(* IEC 61131-3 sources: festo-codesys-mcp/knowledge/library/motion, 4 files *)

(* ---- FB_AxisScaler.st ---- *)
(* =============================================================
   FB_AxisScaler — Axis Unit Conversion (mm/pulses, mm-s/Hz)

   Category:     Motion
   Platform:     CODESYS V3.5 (IEC 61131-3)
   Version:      1.0
   Dependencies: None (standard IEC only)

   Converts between user units (mm, degrees) and machine units
   (encoder pulses, frequency Hz). Handles gear ratio and
   lead screw pitch calculations.

   Usage:
     fbScaler : FB_AxisScaler;
     fbScaler(rPitch := 5.0, nPulsesPerRev := 10000, rGearRatio := 1.0);
     nPulses := fbScaler.fnPosToPulses(rPositionMm := 100.0);
     rMm     := fbScaler.fnPulsesToPos(nPulses := 200000);
   ============================================================= *)
FUNCTION_BLOCK FB_AxisScaler
VAR_INPUT
    rPitch          : REAL := 5.0;         (* Lead screw pitch [mm/rev] or [deg/rev] *)
    nPulsesPerRev   : DINT := 10000;       (* Encoder pulses per revolution *)
    rGearRatio      : REAL := 1.0;         (* Gear ratio (motor/load) *)
END_VAR
VAR_OUTPUT
    rMmPerPulse     : REAL;                (* Conversion factor: mm per pulse *)
    rPulsesPerMm    : REAL;                (* Conversion factor: pulses per mm *)
END_VAR

(* Calculate conversion factors *)
IF nPulsesPerRev > 0 AND ABS(rGearRatio) > 0.0001 THEN
    rMmPerPulse := rPitch / (DINT_TO_REAL(nPulsesPerRev) * rGearRatio);
    IF ABS(rMmPerPulse) > 0.0 THEN
        rPulsesPerMm := 1.0 / rMmPerPulse;
    ELSE
        rPulsesPerMm := 0.0;
    END_IF
ELSE
    rMmPerPulse := 0.0;
    rPulsesPerMm := 0.0;
END_IF

END_FUNCTION_BLOCK

(* ---- FB_BrakeMotor.st ---- *)
(* =============================================================
   FB_BrakeMotor — Motor with Electromagnetic Brake

   Category:     Motion
   Platform:     CODESYS V3.5 (IEC 61131-3)
   Version:      1.0
   Dependencies: None (standard IEC only)

   Controls a motor with electromagnetic holding brake.
   Sequence: Release brake → wait → start motor (and reverse on stop).
   Prevents mechanical shock from simultaneous brake/motor switching.

   Usage:
     fbHoist : FB_BrakeMotor;
     fbHoist(bStart := bCmdHoist, bOverload := bDI_HoistOL);
     bMotorOut := fbHoist.bContactor;
     bBrakeOut := fbHoist.bBrakeRelease;
   ============================================================= *)
FUNCTION_BLOCK FB_BrakeMotor
VAR_INPUT
    bStart          : BOOL;                (* Start command *)
    bOverload       : BOOL := TRUE;        (* Thermal overload (NC) *)
    tBrakeDelay     : TIME := T#300MS;     (* Brake release delay before motor start *)
    tBrakeApply     : TIME := T#200MS;     (* Motor stop delay before brake apply *)
    bEnable         : BOOL := TRUE;        (* Enable control *)
    bReset          : BOOL;                (* Reset error *)
END_VAR
VAR_OUTPUT
    bContactor      : BOOL;                (* Motor contactor output *)
    bBrakeRelease   : BOOL;                (* Brake release output (TRUE=released) *)
    bRunning        : BOOL;                (* Motor is running *)
    bErr          : BOOL;                (* Error active *)
    nErrId          : DINT;                (* 0=OK, 1=Overload *)
END_VAR
VAR
    nState          : INT := 0;
    tonBrakeRel     : TON;
    tonBrakeApp     : TON;
END_VAR

(* Reset *)
IF bReset AND bErr THEN
    nState := 0;
    bErr := FALSE;
    nErrId := 0;
END_IF

(* Overload — immediate stop *)
IF NOT bOverload THEN
    bContactor := FALSE;
    bBrakeRelease := FALSE;
    bRunning := FALSE;
    bErr := TRUE;
    nErrId := 1;
    nState := 10;
    RETURN;
END_IF

IF NOT bEnable THEN
    bContactor := FALSE;
    bBrakeRelease := FALSE;
    bRunning := FALSE;
    nState := 0;
    RETURN;
END_IF

CASE nState OF
0: (* Stopped — brake applied *)
    bContactor := FALSE;
    bBrakeRelease := FALSE;
    bRunning := FALSE;
    tonBrakeRel(IN := FALSE, PT := tBrakeDelay);
    tonBrakeApp(IN := FALSE, PT := tBrakeApply);

    IF bStart THEN
        nState := 1;
    END_IF

1: (* Releasing brake *)
    bBrakeRelease := TRUE;
    bContactor := FALSE;
    tonBrakeRel(IN := TRUE, PT := tBrakeDelay);

    IF tonBrakeRel.Q THEN
        nState := 2;
        tonBrakeRel(IN := FALSE, PT := tBrakeDelay);
    END_IF

    IF NOT bStart THEN
        nState := 0;
        bBrakeRelease := FALSE;
    END_IF

2: (* Running *)
    bContactor := TRUE;
    bBrakeRelease := TRUE;
    bRunning := TRUE;

    IF NOT bStart THEN
        nState := 3;
    END_IF

3: (* Stopping — motor off, brake delayed *)
    bContactor := FALSE;
    bBrakeRelease := TRUE;
    bRunning := FALSE;
    tonBrakeApp(IN := TRUE, PT := tBrakeApply);

    IF tonBrakeApp.Q THEN
        bBrakeRelease := FALSE;
        tonBrakeApp(IN := FALSE, PT := tBrakeApply);
        nState := 0;
    END_IF

10: (* Error *)
    bContactor := FALSE;
    bBrakeRelease := FALSE;
    bRunning := FALSE;

END_CASE

END_FUNCTION_BLOCK

(* ---- FB_StandardMotor.st ---- *)
(* =============================================================
   FB_StandardMotor — Direct-On-Line Motor with Contactor

   Category:     Motion
   Platform:     CODESYS V3.5 (IEC 61131-3)
   Version:      1.0
   Dependencies: None (standard IEC only)

   Controls a standard DOL motor with contactor feedback,
   start delay, and overload protection monitoring.

   Usage:
     fbPump : FB_StandardMotor;
     fbPump(bStart := bCmdPump, bFeedback := bDI_PumpContactor,
            bOverload := bDI_PumpOL);
     bPumpOutput := fbPump.bContactor;
     bPumpRunning := fbPump.bRunning;
   ============================================================= *)
FUNCTION_BLOCK FB_StandardMotor
VAR_INPUT
    bStart          : BOOL;                (* Start command *)
    bFeedback       : BOOL;                (* Contactor feedback (aux contact) *)
    bOverload       : BOOL;                (* Thermal overload relay (NC) *)
    bUseFeedback    : BOOL := FALSE;       (* Enable feedback monitoring *)
    tStartDelay     : TIME := T#0S;        (* Delay before start *)
    tFeedbackTime   : TIME := T#3S;        (* Contactor feedback timeout *)
    bEnable         : BOOL := TRUE;        (* Enable control *)
    bReset          : BOOL;                (* Reset error *)
END_VAR
VAR_OUTPUT
    bContactor      : BOOL;                (* Contactor output *)
    bRunning        : BOOL;                (* Motor is running *)
    bErr          : BOOL;                (* Error active *)
    nErrId          : DINT;                (* 0=OK, 1=Overload, 2=No feedback, 3=Lost feedback *)
END_VAR
VAR
    nState          : INT := 0;
    tonDelay        : TON;
    tonFeedback     : TON;
END_VAR

(* Reset *)
IF bReset AND bErr THEN
    nState := 0;
    bErr := FALSE;
    nErrId := 0;
END_IF

(* Overload trip — immediate stop *)
IF NOT bOverload THEN
    bContactor := FALSE;
    bRunning := FALSE;
    bErr := TRUE;
    nErrId := 1;
    nState := 10;
    RETURN;
END_IF

IF NOT bEnable THEN
    bContactor := FALSE;
    bRunning := FALSE;
    nState := 0;
    RETURN;
END_IF

CASE nState OF
0: (* Stopped *)
    bContactor := FALSE;
    bRunning := FALSE;
    tonDelay(IN := FALSE, PT := tStartDelay);
    tonFeedback(IN := FALSE, PT := tFeedbackTime);

    IF bStart THEN
        nState := 1;
    END_IF

1: (* Start delay *)
    tonDelay(IN := TRUE, PT := tStartDelay);
    IF tonDelay.Q OR tStartDelay = T#0S THEN
        bContactor := TRUE;
        nState := 2;
        tonDelay(IN := FALSE, PT := tStartDelay);
    END_IF

    IF NOT bStart THEN
        nState := 0;
        tonDelay(IN := FALSE, PT := tStartDelay);
    END_IF

2: (* Starting — waiting for feedback *)
    bContactor := TRUE;
    IF bUseFeedback THEN
        tonFeedback(IN := NOT bFeedback, PT := tFeedbackTime);
        IF bFeedback THEN
            bRunning := TRUE;
            nState := 3;
            tonFeedback(IN := FALSE, PT := tFeedbackTime);
        ELSIF tonFeedback.Q THEN
            bContactor := FALSE;
            bErr := TRUE;
            nErrId := 2;
            nState := 10;
        END_IF
    ELSE
        bRunning := TRUE;
        nState := 3;
    END_IF

    IF NOT bStart THEN
        nState := 0;
        bContactor := FALSE;
    END_IF

3: (* Running *)
    bContactor := TRUE;
    bRunning := TRUE;

    (* Lost feedback while running *)
    IF bUseFeedback AND NOT bFeedback THEN
        bContactor := FALSE;
        bRunning := FALSE;
        bErr := TRUE;
        nErrId := 3;
        nState := 10;
    END_IF

    IF NOT bStart THEN
        nState := 0;
        bContactor := FALSE;
        bRunning := FALSE;
    END_IF

10: (* Error *)
    bContactor := FALSE;
    bRunning := FALSE;

END_CASE

END_FUNCTION_BLOCK

(* ---- FB_VfdDrive.st ---- *)
(* =============================================================
   FB_VfdDrive — Variable Frequency Drive Controller

   Category:     Motion
   Platform:     CODESYS V3.5 (IEC 61131-3)
   Version:      1.1
   Dependencies: None (standard IEC only)

   Controls a VFD/inverter via digital outputs (run/direction)
   and analog output (speed reference). Includes ramp limiting,
   fault monitoring, and frequency feedback.

   Festo CMMT-AS/ST Note:
     For Festo servo drives with EtherCAT, use FB_ServoAxis
     with the Festo PtP Package instead. This FB is for
     traditional VFDs controlled via analog/digital I/O.
     See resource: knowledge://festo-ptp-reference

   Usage:
     fbSpindle : FB_VfdDrive;
     fbSpindle(bRun := bCmdSpin, rSpeedRef := 50.0,
               bFault := bDI_VfdFault, nFeedbackHz := nAD_VfdFreq);
     bRunOut   := fbSpindle.bRunOutput;
     nSpeedOut := fbSpindle.nAnalogOut;
   ============================================================= *)
FUNCTION_BLOCK FB_VfdDrive
VAR_INPUT
    bRun            : BOOL;                (* Run command *)
    bReverse        : BOOL;                (* Direction: FALSE=FWD, TRUE=REV *)
    rSpeedRef       : REAL := 0.0;         (* Speed reference [Hz or %] *)
    rSpeedMax       : REAL := 60.0;        (* Maximum speed [Hz] *)
    rRampUpTime     : REAL := 5.0;         (* Acceleration ramp [seconds] *)
    rRampDownTime   : REAL := 3.0;         (* Deceleration ramp [seconds] *)
    bFault          : BOOL;                (* VFD fault input (NO) *)
    nFeedbackHz     : INT := 0;            (* Speed feedback raw [ADC] *)
    nFeedbackMax    : INT := 32767;        (* Feedback at max speed *)
    bEnable         : BOOL := TRUE;        (* Enable control *)
    bReset          : BOOL;                (* Reset error *)
END_VAR
VAR_OUTPUT
    bRunOutput      : BOOL;                (* Run digital output *)
    bDirOutput      : BOOL;                (* Direction output (TRUE=REV) *)
    nAnalogOut      : INT;                 (* Speed ref analog output [0-32767] *)
    rActualSpeed    : REAL;                (* Actual speed [Hz] *)
    bAtSpeed        : BOOL;                (* At target speed (+-2%) *)
    bRunning        : BOOL;                (* Drive is running *)
    bErr          : BOOL;                (* Error active *)
    nErrId          : DINT;                (* 0=OK, 1=VFD fault *)
END_VAR
VAR
    nState          : INT := 0;
    rRampedRef      : REAL := 0.0;
    rRampStep       : REAL;
    rDiff           : REAL;
END_VAR

(* Reset *)
IF bReset AND bErr THEN
    nState := 0;
    bErr := FALSE;
    nErrId := 0;
END_IF

(* VFD fault *)
IF bFault THEN
    bRunOutput := FALSE;
    bRunning := FALSE;
    bErr := TRUE;
    nErrId := 1;
    nState := 10;
END_IF

IF NOT bEnable THEN
    bRunOutput := FALSE;
    bRunning := FALSE;
    rRampedRef := 0.0;
    nState := 0;
END_IF

(* Feedback conversion *)
IF nFeedbackMax > 0 THEN
    rActualSpeed := INT_TO_REAL(nFeedbackHz) / INT_TO_REAL(nFeedbackMax) * rSpeedMax;
ELSE
    rActualSpeed := 0.0;
END_IF

CASE nState OF
0: (* Stopped *)
    bRunOutput := FALSE;
    bRunning := FALSE;
    rRampedRef := 0.0;
    nAnalogOut := 0;

    IF bRun THEN
        bDirOutput := bReverse;
        nState := 1;
    END_IF

1: (* Running — ramping *)
    bRunOutput := TRUE;
    bRunning := TRUE;

    (* Clamp reference *)
    IF rSpeedRef > rSpeedMax THEN rSpeedRef := rSpeedMax; END_IF
    IF rSpeedRef < 0.0 THEN rSpeedRef := 0.0; END_IF

    (* Ramp calculation per scan *)
    rDiff := rSpeedRef - rRampedRef;
    IF rDiff > 0.0 AND rRampUpTime > 0.0 THEN
        rRampStep := rSpeedMax / (rRampUpTime * 1000.0);  (* per ms, approx *)
        rRampedRef := rRampedRef + rRampStep;
        IF rRampedRef > rSpeedRef THEN rRampedRef := rSpeedRef; END_IF
    ELSIF rDiff < 0.0 AND rRampDownTime > 0.0 THEN
        rRampStep := rSpeedMax / (rRampDownTime * 1000.0);
        rRampedRef := rRampedRef - rRampStep;
        IF rRampedRef < rSpeedRef THEN rRampedRef := rSpeedRef; END_IF
    ELSE
        rRampedRef := rSpeedRef;
    END_IF

    (* Convert to analog output *)
    IF rSpeedMax > 0.0 THEN
        nAnalogOut := REAL_TO_INT(rRampedRef / rSpeedMax * 32767.0);
    ELSE
        nAnalogOut := 0;
    END_IF
    IF nAnalogOut < 0 THEN nAnalogOut := 0; END_IF
    IF nAnalogOut > 32767 THEN nAnalogOut := 32767; END_IF

    (* At speed detection *)
    bAtSpeed := ABS(rRampedRef - rSpeedRef) < (rSpeedMax * 0.02);

    IF NOT bRun THEN
        nState := 2;
    END_IF

2: (* Decelerating to stop *)
    bRunning := TRUE;
    IF rRampDownTime > 0.0 THEN
        rRampStep := rSpeedMax / (rRampDownTime * 1000.0);
        rRampedRef := rRampedRef - rRampStep;
    END_IF
    IF rRampedRef <= 0.0 THEN
        rRampedRef := 0.0;
        nState := 0;
    END_IF
    IF rSpeedMax > 0.0 THEN
        nAnalogOut := REAL_TO_INT(rRampedRef / rSpeedMax * 32767.0);
    ELSE
        nAnalogOut := 0;
    END_IF
    IF nAnalogOut < 0 THEN nAnalogOut := 0; END_IF
    bAtSpeed := FALSE;

10: (* Error *)
    bRunOutput := FALSE;
    bRunning := FALSE;
    rRampedRef := 0.0;
    nAnalogOut := 0;

END_CASE

END_FUNCTION_BLOCK
